// TIA Portal project "UDT_kullanici_tanimli_data tipi olusturma" (V18)

(* hardware
DEVICE "S7-1200 station_1"  S7-1200 Station
   slot 0: "Rack_0"  S7-1200 Rack  Rack  V1.0
   slot 1: "PLC_1"  CPU 1214C DC/DC/DC  6ES7 214-1AG40-0XB0  V4.6
*)

// ===== PLC "PLC_1"  CPU 1214C DC/DC/DC =====

TYPE "KAZAN"
   STRUCT
      DOLDURMA : Bool;
      BOŞALTMA : Bool;
      KARIŞTIRMA : Bool;
      SEVİYE : Int := 50;
      SICAKLIK : Int := 60;
   END_STRUCT;
END_TYPE

DATA_BLOCK "KAZANLAR"   // DB1
{ S7_Optimized_Access := 'TRUE' }
VERSION : 0.1
   VAR
      KAZAN1 : "KAZAN";
      KAZAN2 : "KAZAN";
      KAZAN3 : "KAZAN";
   END_VAR
BEGIN
END_DATA_BLOCK

ORGANIZATION_BLOCK "Main"   // OB1, LAD, ProgramCycle
TITLE = "Main Program Sweep (Cycle)"
{ S7_Optimized_Access := 'TRUE' }
VERSION : 0.1
   VAR_INPUT
      Initial_Call : Bool;   // Initial call of this OB
      Remanence : Bool;   // =True, if remanent data are available
   END_VAR
BEGIN

REGION Network 1
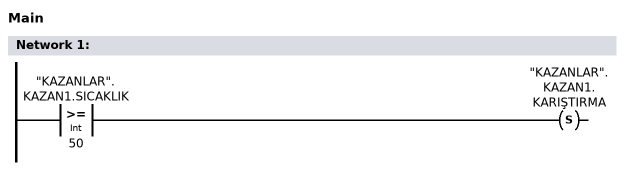
   RUNG wire#powerrail
      { S7_Templates := "SrcType := Int" } GE_Contact(in1 := "KAZANLAR".KAZAN1.SICAKLIK, in2 := 50)
      S_Coil( "KAZANLAR".KAZAN1.KARIŞTIRMA )
   END_RUNG
   // the same network as SCL:
   IF "KAZANLAR".KAZAN1.SICAKLIK >= 50 THEN "KAZANLAR".KAZAN1.KARIŞTIRMA := TRUE; END_IF;
END_REGION
END_ORGANIZATION_BLOCK